PROGRAM P_Demo_F_ULARGE
VAR
    ulgLargeAccum : T_ULARGE_INTEGER; // 业务量（T_ULARGE_INTEGER）
    bPackArg      : BOOL; // 在线置 TRUE 触发一次打包
    argDescriptor : T_Arg; // 打包后的 T_Arg 描述符（含 eType/cbLen/pData）
END_VAR

// ============================================================
// Tc2_Utilities.F_ULARGE 演示程序（FUNCTION，返回 T_Arg）
// ============================================================
// 场景：把 T_ULARGE_INTEGER 业务量打包为 T_Arg，供下游 EventLogger / FormatString2
//       / ADS 消息的可变参数机制使用。
// 价值：替代手填 T_Arg 三字段（eType/cbLen/pData），一行调用搞定。
// 验证：在线写 ulgLargeAccum 为示例值，bPackArg := TRUE；
//       下一周期 argDescriptor.cbLen = SIZEOF(T_ULARGE_INTEGER)，argDescriptor.pData <> 0。
// ============================================================

IF bPackArg THEN
    // 单次完整调用：返回的 T_Arg 立即可喂给 F_PutInArg(arg := argDescriptor, ...)
    argDescriptor := F_ULARGE(ulgLargeAccum);
    bPackArg := FALSE;
END_IF;

END_PROGRAM

(* stored: Version 1.1.0.1, ProductVersion 3.1.4024.5
   POU P_Demo_F_ULARGE: Id {4a6fcf25-9223-52ad-892d-e3e1af4406cc}, SpecialFunc None *)
